FUNCTION_BLOCK FB_ADS_Comm
VAR_INPUT
	bEnable				: BOOL;			// TRUE to run communication
	eType				: E_ADS_Comm_Type;// Read or write
	rInterval			: REAL;			// Update interval [s]
	pLocalVar			: PVOID;		// Pointer to local variable to link to remote device
	nLocalSize			: UINT;			// Size of local variable
	sNetID				: T_AmsNetId;	// ADS address on remote ADS device
	nPort				: T_AmsPort;	// ADS port on remote ADS device
	sVarName			: STRING;		// Remote symbol name to read/write
END_VAR
VAR_OUTPUT
	bWriteError			: BOOL;			// Writing error
	bReadError			: BOOL;			// Reading error
	bParameterError		: BOOL;			// Parameter error
END_VAR
VAR
	fbReadAds			: FB_ReadAdsSymByName;	// FB to read symbols via. ADS
	fbWriteAds 			: FB_WriteAdsSymByName;	// FB to write symbols via. ADS
	nState				: E_ADS_Comm_State;		// State
	tonExecute			: TON;					// Execute timer
	tonInterval			: TON;					// For calculating actual read/write interval
	rActInterval		: REAL;					// [s] Measured read/write interval
	bSendRecv			: BOOL;					// TRUE to read or write data
	bSendRecvDone		: BOOL;					// TRUE when completed
END_VAR

IF (bEnable) THEN
	// Check parameters
	IF (sNetID = '') THEN
		bParameterError := TRUE;
	ELSIF (nPort = 0) THEN
		bParameterError := TRUE;
	ELSIF (pLocalVar = 0) THEN
		bParameterError := TRUE;
	ELSIF (nLocalSize <= 0) THEN
		bParameterError := TRUE;
	ELSE
		bParameterError := FALSE;
	END_IF
ELSE
	bParameterError := FALSE;
	bReadError := FALSE;
	bWriteError := FALSE;
	bSendRecvDone := FALSE;
END_IF

// Check interval
IF (rInterval < 0) THEN
	rInterval := 0;
END_IF

// Run read FB
IF (bEnable) THEN
	// ADS communication
	CASE nState OF
		E_ADS_Comm_State.Disabled:
			bWriteError := FALSE;
			bReadError := FALSE;
			bParameterError := FALSE;
			tonExecute.IN := FALSE;
			fbReadAds.bRead := FALSE;
			fbWriteAds.bWrite := FALSE;
			IF (bEnable) THEN
				nState := E_ADS_Comm_State.Idle;
			END_IF

		E_ADS_Comm_State.Idle:
			tonExecute.IN := TRUE;
			IF (NOT bEnable) THEN
				nState := E_ADS_Comm_State.Disabled;
			ELSIF (eType = ADS_RD_FAST) THEN
				nState := E_ADS_Comm_State.Wait_Read;
			ELSIF (eType = ADS_WR_FAST) THEN
				nState := E_ADS_Comm_State.Wait_Write;
			ELSIF (eType = ADS_RD_SLOW) THEN
				nState := E_ADS_Comm_State.Wait_Read;
			ELSIF (eType = ADS_WR_SLOW) THEN
				nState := E_ADS_Comm_State.Wait_Write;
			ELSIF (eType = ADS_WR_TRIG1) THEN
				nState := E_ADS_Comm_State.Wait_Write;
			ELSIF (eType = ADS_WR_TRIG2) THEN
				nState := E_ADS_Comm_State.Wait_Write;
			ELSIF (eType = ADS_WR_TRIG3) THEN
				nState := E_ADS_Comm_State.Wait_Write;
			END_IF

		E_ADS_Comm_State.Wait_Write:
			IF (tonExecute.Q OR bSendRecv) THEN
				tonExecute.IN := FALSE;
				fbWriteAds.bWrite := TRUE;
				fbWriteAds.sNetID := sNetID; 
				fbWriteAds.nPort := nPort; 
				fbWriteAds.sVarName := sVarName; 
				fbWriteAds.nSrcAddr := pLocalVar;
				fbWriteAds.nLen := nLocalSize;
//				fbWriteAds.eComMode := eAdsComModeFastCom;
				fbWriteAds.eComMode := eAdsComModeSecureCom;
				nState := E_ADS_Comm_State.Writing;		
			END_IF

		E_ADS_Comm_State.Writing:
			IF (fbWriteAds.bBusy) THEN
				tonExecute.IN := TRUE;
			ELSE
				fbWriteAds.bWrite := FALSE;
				IF (fbWriteAds.bError) THEN
					nState := E_ADS_Comm_State.Write_Error;
				ELSE
					rActInterval := (TIME_TO_REAL(tonInterval.ET) / 1000.0);
					tonInterval(IN := FALSE);
					bWriteError := FALSE;
					bSendRecvDone := TRUE;
					nState := E_ADS_Comm_State.Idle;
				END_IF
			END_IF

		E_ADS_Comm_State.Write_Error:
			bWriteError := TRUE;		
			nState := E_ADS_Comm_State.Idle;

		E_ADS_Comm_State.Wait_Read:
			IF (tonExecute.Q OR bSendRecv) THEN
				tonExecute.IN := FALSE;
				fbReadAds.bRead := TRUE;
				fbReadAds.sNetID := sNetID;
				fbReadAds.nPort := nPort; 
				fbReadAds.sVarName := sVarName; 
				fbReadAds.nDestAddr := pLocalVar;
				fbReadAds.nLen := nLocalSize;
//				fbReadAds.eComMode := eAdsComModeFastCom;
				fbReadAds.eComMode := eAdsComModeSecureCom;
				nState := E_ADS_Comm_State.Reading;	
			END_IF

		E_ADS_Comm_State.Reading:
			IF (fbReadAds.bBusy) THEN
				tonExecute.IN := TRUE;
			ELSE
				fbReadAds.bRead := FALSE;
				IF (fbReadAds.bError) THEN
					nState := E_ADS_Comm_State.Read_Error;
				ELSE
					rActInterval := (TIME_TO_REAL(tonInterval.ET) / 1000.0);
					tonInterval(IN := FALSE);
					bReadError := FALSE;
					bSendRecvDone := TRUE;
					nState := E_ADS_Comm_State.Idle;
				END_IF
			END_IF
		
		E_ADS_Comm_State.Read_Error:
			bReadError := TRUE;		
			nState := E_ADS_Comm_State.Idle;

		ELSE
			nState := E_ADS_Comm_State.Disabled;
	END_CASE

	IF ((eType = ADS_WR_TRIG1) OR (eType = ADS_WR_TRIG2) OR (eType = ADS_WR_TRIG3) OR
		(eType = ADS_RD_TRIG1) OR (eType = ADS_RD_TRIG2) OR (eType = ADS_RD_TRIG3)) THEN
		// No cyclic reading/writing
		tonExecute.IN := FALSE;
	END_IF
	tonExecute.PT := REAL_TO_TIME(rInterval * 1000.0);
	tonExecute();
	tonInterval(IN := TRUE, PT := T#60S);
	fbReadAds.tTimeout := DEFAULT_ADS_TIMEOUT;
	fbReadAds();
	fbWriteAds();
	fbWriteAds.tTimeout := DEFAULT_ADS_TIMEOUT;

END_IF

METHOD PUBLIC M_SendRecv : BOOL
VAR_INPUT
END_VAR
IF ((eType = E_ADS_Comm_Type.ADS_WR_TRIG1) OR (eType = E_ADS_Comm_Type.ADS_RD_TRIG1) OR
	(eType = E_ADS_Comm_Type.ADS_WR_TRIG2) OR (eType = E_ADS_Comm_Type.ADS_RD_TRIG2) OR
	(eType = E_ADS_Comm_Type.ADS_WR_TRIG3) OR (eType = E_ADS_Comm_Type.ADS_RD_TRIG3)) THEN
	
	IF (NOT bSendRecv) THEN
		bSendRecvDone := FALSE;	
	END_IF
	bSendRecv := TRUE;
END_IF
END_METHOD

METHOD PUBLIC M_SendRecvCompleted : BOOL
VAR_INPUT
END_VAR
M_SendRecvCompleted := bSendRecvDone;
END_METHOD

METHOD PUBLIC M_SendRecvStop : BOOL
VAR_INPUT
END_VAR
bSendRecv := FALSE;
END_METHOD

END_FUNCTION_BLOCK

(* stored: Version 1.1.0.1, ProductVersion 3.1.4024.2
   POU FB_ADS_Comm: Id {bbf34da6-337f-4ae0-9a1f-743a6b51d4fb}, SpecialFunc None
   Method M_SendRecv: Id {009253eb-80af-48d0-ba2c-2cc257cb53b8}
   Method M_SendRecvCompleted: Id {ea8cecad-8b25-47cf-8a5b-b80c4b123c02}
   Method M_SendRecvStop: Id {831511df-6d2a-4548-8ab4-b6c88da194a6} *)
